// TIA Portal V20 export
DATA_BLOCK "CS_MOVIKIT"   // DB28
{ S7_Optimized_Access := 'TRUE' }
// stored: MemoryReserve 100
   VAR
      CS_RL_PI : "SEW_MOVIKIT_VelocityDrive_STATUS_V2.1";
      CS_RL_PO : "SEW_MOVIKIT_VelocityDrive_SETPOINTS_V2.1";
      CS_RP_PI : "SEW_MOVIKIT_VelocityDrive_STATUS_V2.1";
      CS_RP_PO : "SEW_MOVIKIT_VelocityDrive_SETPOINTS_V2.1";
      CS_M1_PI : "SEW_MOVIKIT_VelocityDrive_STATUS_V2.1";
      CS_M1_PO : "SEW_MOVIKIT_VelocityDrive_SETPOINTS_V2.1";
      CS_M2_PI : "SEW_MOVIKIT_VelocityDrive_STATUS_V2.1";
      CS_M2_PO : "SEW_MOVIKIT_VelocityDrive_SETPOINTS_V2.1";
   END_VAR
BEGIN
END_DATA_BLOCK
